(* CODESYS project TrabalhoFMSLadder.project

Project tree, tasks and I/O mapping:
  Device : CODESYS Control Win V3, 3S - Smart Software Solutions GmbH, order no. 305021, version 3.5.11.30
    application Application
      libraries: Standard, * (System); EA_XiocEvents, 3.5.2.0 (Eaton Automation); Standard64, * (System); Util, * (System)
      task MainTask (cyclic, interval t#20ms, priority 1) calls LinhaFabricacao, LinhaEntradaTampa, RobosDaora, LinhaSaidaUsinagem, EstacaoTampa, Armazenamento, SaidaPecas, EstacaoPallet
      Symbols
      program LinhaFabricacao [LD]
      program LinhaEntradaTampa [LD]
      program RobosDaora [LD]
      program LinhaSaidaUsinagem [LD]
      program EstacaoTampa [LD]
      program Armazenamento [LD]
      program SaidaPecas [LD]
      program EstacaoPallet [LD]
      program Teste [LD]
  program PLC_PRG_1 [LD]
  program PLC_PRG [LD]
  program PLC_PRG_2 [LD]
*)

// Device/Application/LinhaFabricacao
PROGRAM LinhaFabricacao
VAR
		//ENTRADAS
	SensorDifuso1CLP:BOOL;
	SensorDifuso2CLP:BOOL;
	VisionSensor1CLP:BOOL;
	VisionSensor2CLP:BOOL;
	ConveyorGate1OpenCLP:BOOL;
	
	//Saidas
	StopBlade1CLP:BOOL;
	StopBlade2CLP:BOOL;
	Pusher1CLP:BOOL;
	Pusher2CLP:BOOL;
	ConveyorGate1CLP:BOOL;
	Conveyor6m1CLP:BOOL;
	Conveyor6m2CLP:BOOL;
	
	
	//Memórias
	Conv6m1Vazio:BOOL;
	Conv6m2Vazio:BOOL;
	TravaVerde:BOOL;
	TravaAzul:BOOL;
	LerVerde: BOOL;
	LerAzul: BOOL;
	RejeitadoVerde:BOOL;
	RejeitadoAzul:BOOL;
	
	//vars timers
	ElapsedTime: TIME;
	ElapsedTime2: TIME;
	TimerVerde: TON;
	TimerAzul: TON;
	TimerPusher1: TON;
	TimerPusher2: TON;
END_VAR
VAR // added by the converter: edge detectors and wires of the graphical bodies
    _w1, _w2 : BOOL;
END_VAR

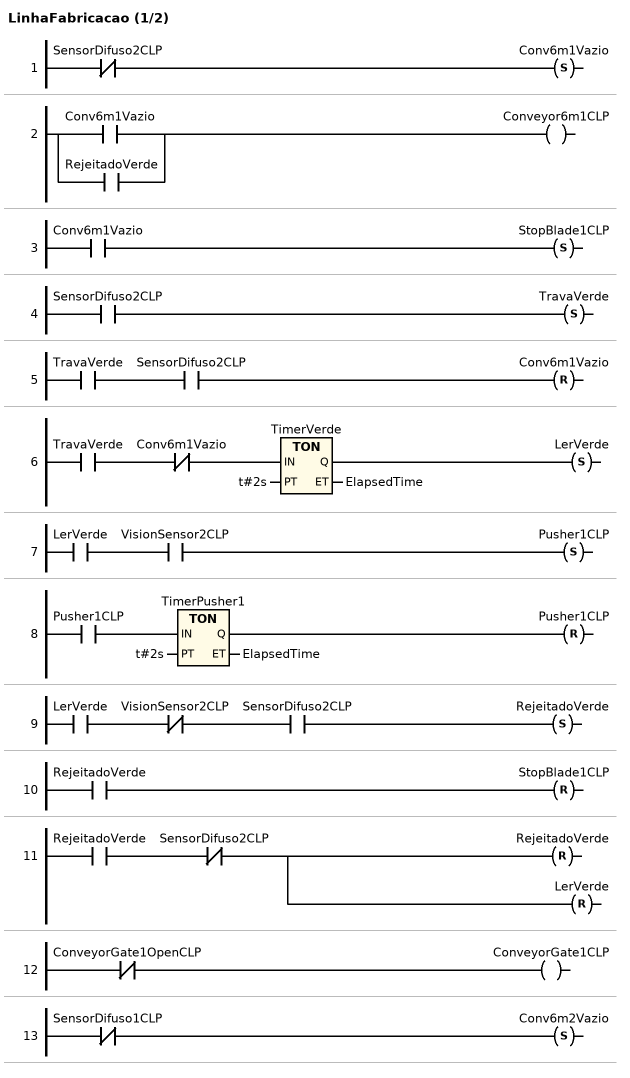
// NETWORK 1
Conv6m1Vazio S= NOT SensorDifuso2CLP;

// NETWORK 2
Conveyor6m1CLP := Conv6m1Vazio OR RejeitadoVerde;

// NETWORK 3
StopBlade1CLP S= Conv6m1Vazio;

// NETWORK 4
TravaVerde S= SensorDifuso2CLP;

// NETWORK 5
Conv6m1Vazio R= TravaVerde AND SensorDifuso2CLP;

// NETWORK 6
TimerVerde(IN := TravaVerde AND NOT Conv6m1Vazio, PT := t#2s, ET => ElapsedTime); // TON
LerVerde S= TimerVerde.Q;

// NETWORK 7
Pusher1CLP S= LerVerde AND VisionSensor2CLP;

// NETWORK 8
TimerPusher1(IN := Pusher1CLP, PT := t#2s, ET => ElapsedTime); // TON
Pusher1CLP R= TimerPusher1.Q;

// NETWORK 9
RejeitadoVerde S= LerVerde AND NOT VisionSensor2CLP AND SensorDifuso2CLP;

// NETWORK 10
StopBlade1CLP R= RejeitadoVerde;

// NETWORK 11
_w1 := RejeitadoVerde AND NOT SensorDifuso2CLP;
RejeitadoVerde R= _w1;
LerVerde R= _w1;

// NETWORK 12
ConveyorGate1CLP := NOT ConveyorGate1OpenCLP;

// NETWORK 13
Conv6m2Vazio S= NOT SensorDifuso1CLP;

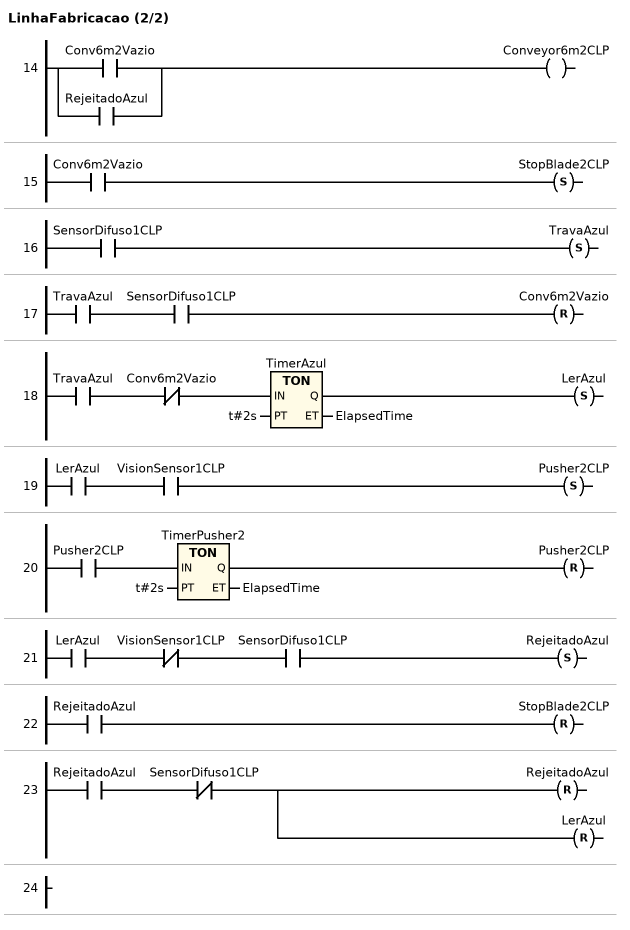
// NETWORK 14
Conveyor6m2CLP := Conv6m2Vazio OR RejeitadoAzul;

// NETWORK 15
StopBlade2CLP S= Conv6m2Vazio;

// NETWORK 16
TravaAzul S= SensorDifuso1CLP;

// NETWORK 17
Conv6m2Vazio R= TravaAzul AND SensorDifuso1CLP;

// NETWORK 18
TimerAzul(IN := TravaAzul AND NOT Conv6m2Vazio, PT := t#2s, ET => ElapsedTime); // TON
LerAzul S= TimerAzul.Q;

// NETWORK 19
Pusher2CLP S= LerAzul AND VisionSensor1CLP;

// NETWORK 20
TimerPusher2(IN := Pusher2CLP, PT := t#2s, ET => ElapsedTime); // TON
Pusher2CLP R= TimerPusher2.Q;

// NETWORK 21
RejeitadoAzul S= LerAzul AND NOT VisionSensor1CLP AND SensorDifuso1CLP;

// NETWORK 22
StopBlade2CLP R= RejeitadoAzul;

// NETWORK 23
_w2 := RejeitadoAzul AND NOT SensorDifuso1CLP;
RejeitadoAzul R= _w2;
LerAzul R= _w2;

// NETWORK 24

END_PROGRAM

// Device/Application/LinhaEntradaTampa
PROGRAM LinhaEntradaTampa
VAR
	//entradas
	VisionSensor3CLP:BOOL;
	SensorDifuso6CLP:BOOL;
	SensorDifuso7CLP:BOOL;
	
	//saidas
	Conveyor6m3CLP:BOOL;
	Conveyor4m1CLP:BOOL;
	ArmSorterCLP:BOOL;
	ArmBeltCLP:BOOL;
	Emmiter3CLP:BOOL;
	
	//memorias
	DivAzul:BOOL;
	TimerDiv: TON;
	Tempodiv: TIME;
	TimerDivR: TON;

	TesteCLP: BOOL;
	Nada: BOOL;
	StopBlade5CLP: BOOL;
	StopBlade6CLP: BOOL;
END_VAR

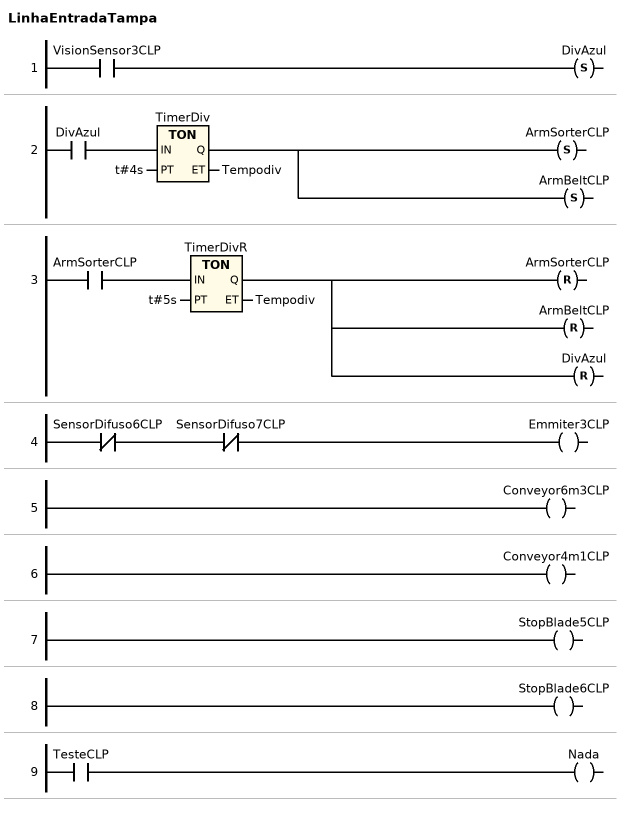
// NETWORK 1
DivAzul S= VisionSensor3CLP;

// NETWORK 2
TimerDiv(IN := DivAzul, PT := t#4s, ET => Tempodiv); // TON
ArmSorterCLP S= TimerDiv.Q;
ArmBeltCLP S= TimerDiv.Q;

// NETWORK 3
TimerDivR(IN := ArmSorterCLP, PT := t#5s, ET => Tempodiv); // TON
ArmSorterCLP R= TimerDivR.Q;
ArmBeltCLP R= TimerDivR.Q;
DivAzul R= TimerDivR.Q;

// NETWORK 4
Emmiter3CLP := NOT SensorDifuso6CLP AND NOT SensorDifuso7CLP;

// NETWORK 5
Conveyor6m3CLP := TRUE;

// NETWORK 6
Conveyor4m1CLP := TRUE;

// NETWORK 7
StopBlade5CLP := TRUE;

// NETWORK 8
StopBlade6CLP := TRUE;

// NETWORK 9
Nada := TesteCLP;

END_PROGRAM

// Device/Application/RobosDaora
PROGRAM RobosDaora
VAR
	//saidas
	MachinigCenter1StartCLP:BOOL;
	MachinigCenter2StartCLP:BOOL;
	MachinigCenter1StopCLP:BOOL;
	MachinigCenter2StopCLP:BOOL;
	MachinigCenter1ResetCLP:BOOL;
	MachinigCenter2ResetCLP:BOOL;

	//memorias
	InitialStart: TP;
	timepulse: TIME;
	BotaoSupLiga1:BOOL;
	BotaoSupLiga2:BOOL;
	BotaoSupPara1:BOOL;
	BotaoSupPara2:BOOL;
	BotaoSupReset1:BOOL;
	BotaoSupReset2:BOOL;
	
	//fb
	Progress1CLP: INT;
	Nada: BOOL;
	FDS1: INT;
	Progress2CLP: INT;
	FDS2: INT;
	Start1CLP: BOOL;
	Start2CLP: BOOL;
	Stop1CLP: BOOL;
	Stop2CLP: BOOL;
	Open1CLP: BOOL;
	Open2CLP: BOOL;
END_VAR

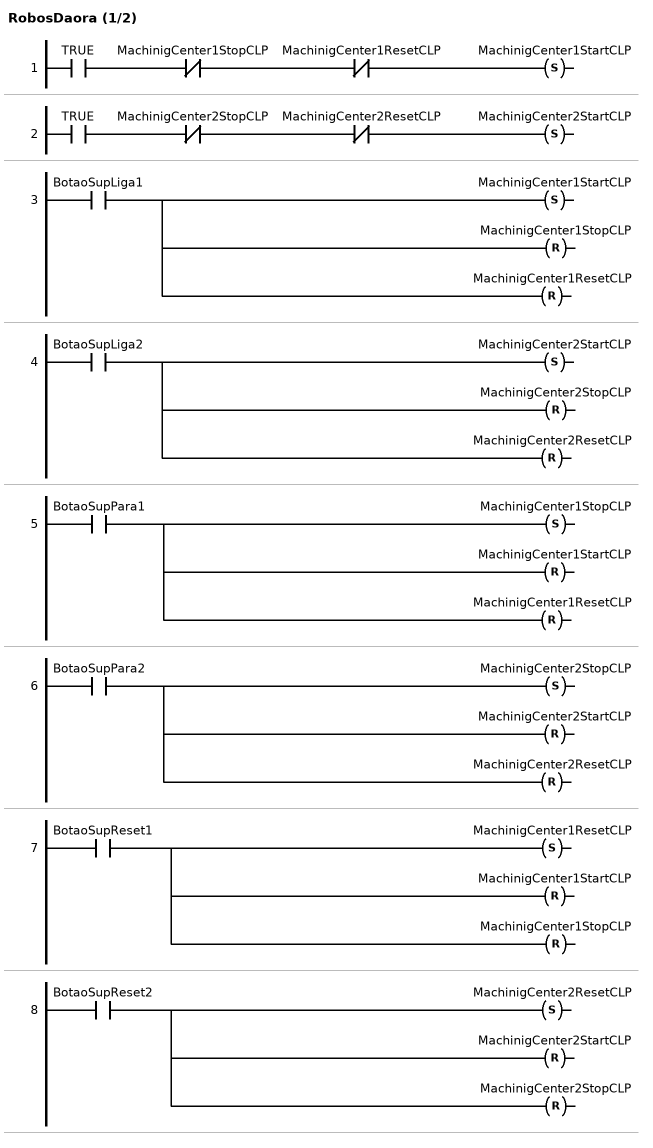
// NETWORK 1
MachinigCenter1StartCLP S= TRUE AND NOT MachinigCenter1StopCLP AND NOT MachinigCenter1ResetCLP;

// NETWORK 2
MachinigCenter2StartCLP S= TRUE AND NOT MachinigCenter2StopCLP AND NOT MachinigCenter2ResetCLP;

// NETWORK 3
MachinigCenter1StartCLP S= BotaoSupLiga1;
MachinigCenter1StopCLP R= BotaoSupLiga1;
MachinigCenter1ResetCLP R= BotaoSupLiga1;

// NETWORK 4
MachinigCenter2StartCLP S= BotaoSupLiga2;
MachinigCenter2StopCLP R= BotaoSupLiga2;
MachinigCenter2ResetCLP R= BotaoSupLiga2;

// NETWORK 5
MachinigCenter1StopCLP S= BotaoSupPara1;
MachinigCenter1StartCLP R= BotaoSupPara1;
MachinigCenter1ResetCLP R= BotaoSupPara1;

// NETWORK 6
MachinigCenter2StopCLP S= BotaoSupPara2;
MachinigCenter2StartCLP R= BotaoSupPara2;
MachinigCenter2ResetCLP R= BotaoSupPara2;

// NETWORK 7
MachinigCenter1ResetCLP S= BotaoSupReset1;
MachinigCenter1StartCLP R= BotaoSupReset1;
MachinigCenter1StopCLP R= BotaoSupReset1;

// NETWORK 8
MachinigCenter2ResetCLP S= BotaoSupReset2;
MachinigCenter2StartCLP R= BotaoSupReset2;
MachinigCenter2StopCLP R= BotaoSupReset2;

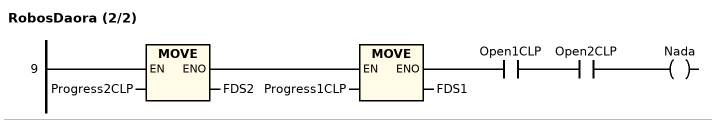
// NETWORK 9
FDS2 := Progress2CLP;
FDS1 := Progress1CLP;
Nada := Open1CLP AND Open2CLP;

END_PROGRAM

// Device/Application/LinhaSaidaUsinagem
PROGRAM LinhaSaidaUsinagem
VAR
	//SAIDAS
	EsteiraUsinada1CLP:BOOL;
	EsteiraPortaoUsinadaCLP:BOOL;
	Conveyor4m2CLP:BOOL;
	Conveyor2m1CLP:BOOL;
	StopBlade7CLP:BOOL;
	
	//ENTRADAS
	SensorDifuso5CLP:BOOL;
	PortaoUsinadaOpenCLP:BOOL;
	
	//Memórias
	EsteirasON:BOOL;
	PecaDentro:BOOL;
	PecaNoSensor:BOOL;
END_VAR
VAR // added by the converter: edge detectors and wires of the graphical bodies
    _w1, _w2 : BOOL;
END_VAR

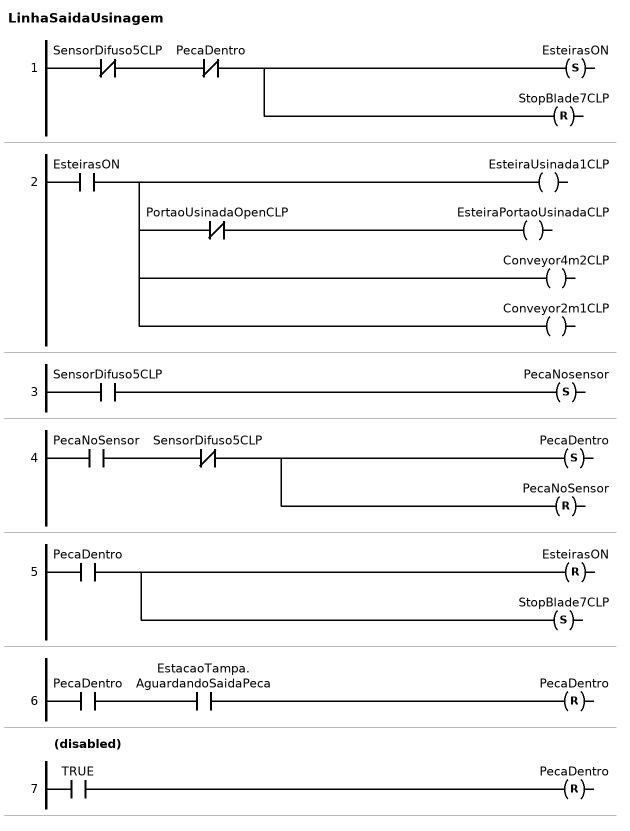
// NETWORK 1
_w1 := NOT SensorDifuso5CLP AND NOT PecaDentro;
EsteirasON S= _w1;
StopBlade7CLP R= _w1;

// NETWORK 2
EsteiraUsinada1CLP := EsteirasON;
EsteiraPortaoUsinadaCLP := EsteirasON AND NOT PortaoUsinadaOpenCLP;
Conveyor4m2CLP := EsteirasON;
Conveyor2m1CLP := EsteirasON;

// NETWORK 3
PecaNosensor S= SensorDifuso5CLP;

// NETWORK 4
_w2 := PecaNoSensor AND NOT SensorDifuso5CLP;
PecaDentro S= _w2;
PecaNoSensor R= _w2;

// NETWORK 5
EsteirasON R= PecaDentro;
StopBlade7CLP S= PecaDentro;

// NETWORK 6
PecaDentro R= PecaDentro AND EstacaoTampa.AguardandoSaidaPeca;

// NETWORK 7 (disabled)
// PecaDentro R= TRUE;

END_PROGRAM

// Device/Application/EstacaoTampa
PROGRAM EstacaoTampa
VAR
	//SAIDAS
	Conveyor2m3CLP:BOOL;
	StopBlade4CLP:BOOL;
	Pick1XSetPointCLP:LREAL;
	Pick1YSetPointCLP:LREAL;
	Pick1ZSetPointCLP:LREAL;
	Pick1GrabCLP:BOOL;
	//ENTRADAS
	PickSensorCLP:BOOL;
	VisionSensor4_0CLP:BOOL;
	VisionSensor4_1CLP:BOOL;
	VisionSensor4_2CLP:BOOL;
	
	//MEMORIAS
	EsteiraON:BOOL;
	VerCor:BOOL;
	PegaAzul:BOOL;
	PegaVerde:BOOL;
	AvancaTampa:BOOL;
	PegaTampa:BOOL;
	RecuaGraber:BOOL;
	GraberRecuado:BOOL;
	TampaPegada:BOOL;
	ColetaTampa:BOOL;
	ColocarTampa:BOOL;
	TampaPosicionada:BOOL;
	SoltaTampa:BOOL;
	PosicaoDescanso:BOOL;
	RetornoPosInicial:BOOL;
	LiberarPeca:BOOL;
	AguardandoSaidaPeca:BOOL;
	EstacaoOcupada:BOOL;
	
	TimerMove1: TON;
	ElapsedTime1: TIME;
	TimerPegar: TON;
	ElapsedTime2: TIME;
	TimerRecuo: TON;
	TimerMove2: TON;
	TimerWait: TON;
	ElapsedTime3: TIME;
	ElapsedTime4: TIME;
	ElapsedTime5: TIME;
	ElapsedTime6: TIME;
	ElapsedTIme7: TIME;
	TimerRecuo2: TON;
	TimerMove3: TON;
	TimerSoltar: TON;
	ElapsedTime8: TIME;
	TimerSaida: TON;
	ElapsedTime9: TIME;
	TimerWait2: TON;
	ElapsedTIme10: TIME;
	TimerWait3: TON;
	ElapsedTime11: TIME;
END_VAR
VAR // added by the converter: edge detectors and wires of the graphical bodies
    _w1, _w2, _w3, _w4, _w5, _w6, _w7, _w8, _w9, _w10, _w11, _w12 : BOOL;
END_VAR

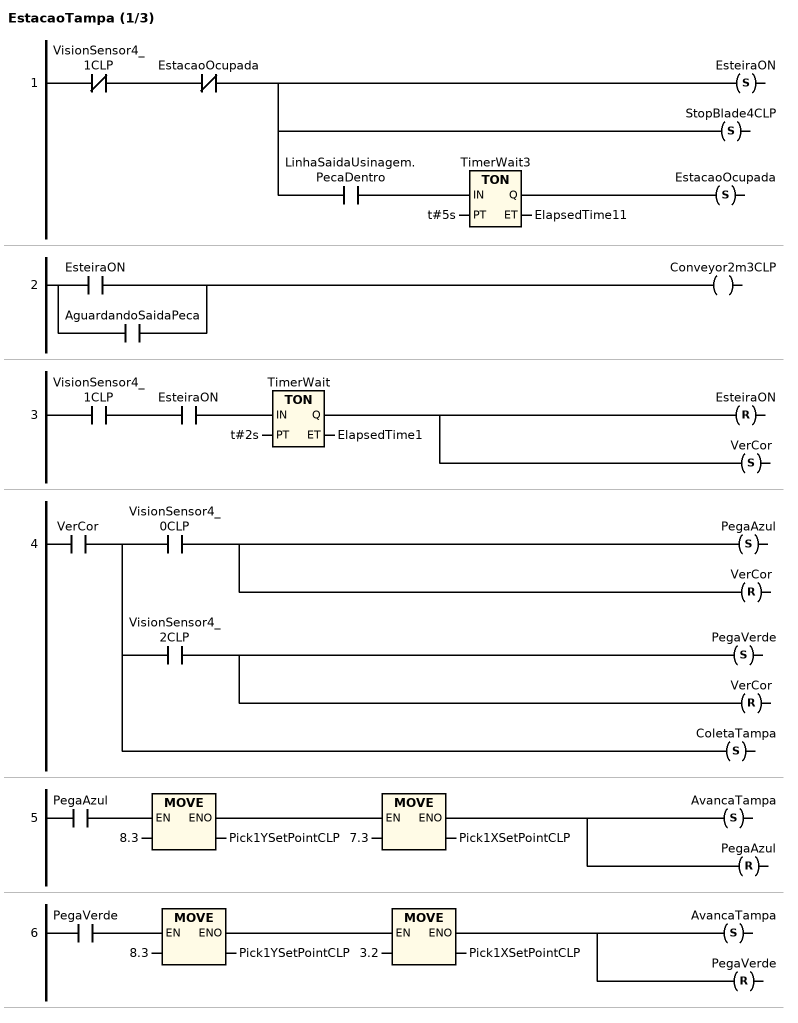
// NETWORK 1
_w1 := NOT VisionSensor4_1CLP AND NOT EstacaoOcupada;
EsteiraON S= _w1;
StopBlade4CLP S= _w1;
TimerWait3(IN := _w1 AND LinhaSaidaUsinagem.PecaDentro, PT := t#5s, ET => ElapsedTime11); // TON
EstacaoOcupada S= TimerWait3.Q;

// NETWORK 2
Conveyor2m3CLP := EsteiraON OR AguardandoSaidaPeca;

// NETWORK 3
TimerWait(IN := VisionSensor4_1CLP AND EsteiraON, PT := t#2s, ET => ElapsedTime1); // TON
EsteiraON R= TimerWait.Q;
VerCor S= TimerWait.Q;

// NETWORK 4
_w2 := VerCor;
_w3 := _w2 AND VisionSensor4_0CLP;
PegaAzul S= _w3;
VerCor R= _w3;
_w4 := _w2 AND VisionSensor4_2CLP;
PegaVerde S= _w4;
VerCor R= _w4;
ColetaTampa S= _w2;

// NETWORK 5
_w5 := PegaAzul;
IF _w5 THEN Pick1YSetPointCLP := 8.3; END_IF
IF _w5 THEN Pick1XSetPointCLP := 7.3; END_IF
AvancaTampa S= _w5;
PegaAzul R= _w5;

// NETWORK 6
_w6 := PegaVerde;
IF _w6 THEN Pick1YSetPointCLP := 8.3; END_IF
IF _w6 THEN Pick1XSetPointCLP := 3.2; END_IF
AvancaTampa S= _w6;
PegaVerde R= _w6;

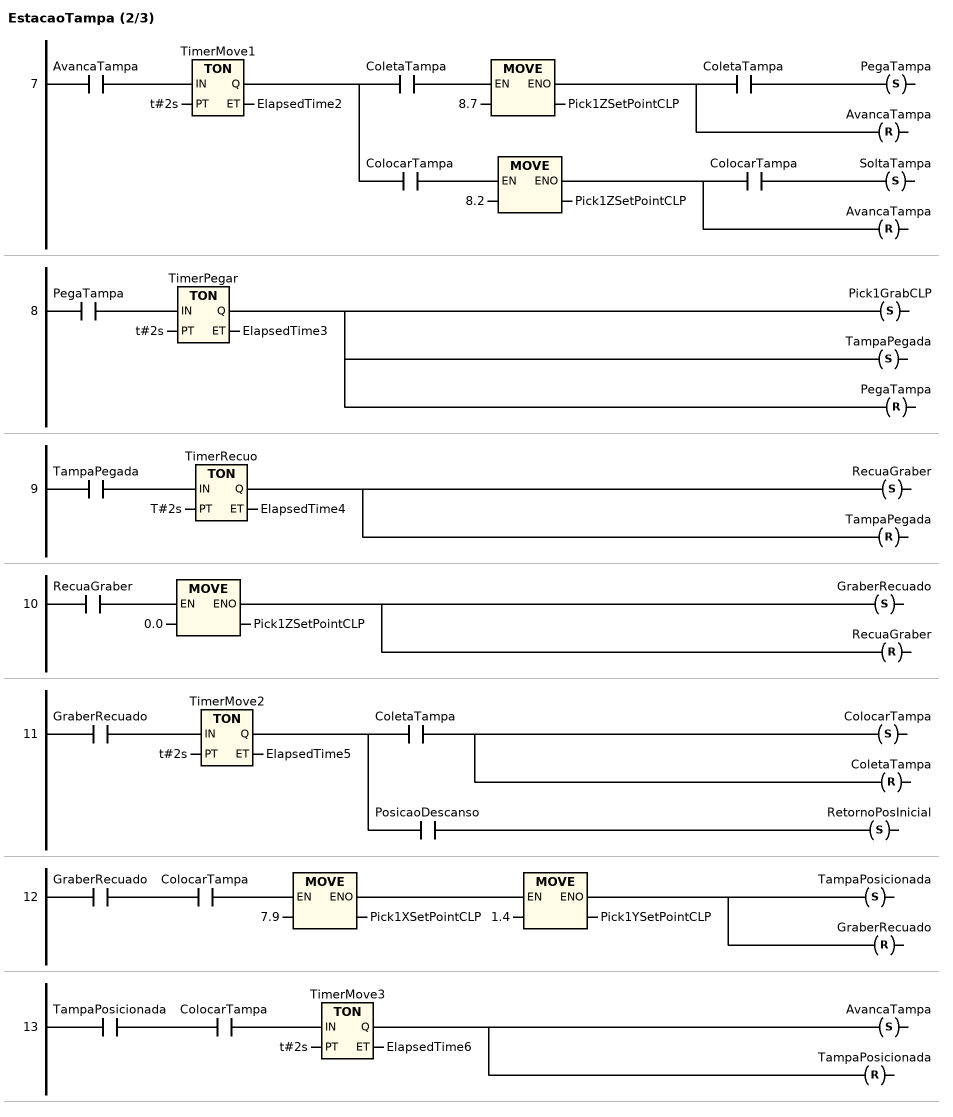
// NETWORK 7
TimerMove1(IN := AvancaTampa, PT := t#2s, ET => ElapsedTime2); // TON
_w7 := TimerMove1.Q AND ColetaTampa;
IF _w7 THEN Pick1ZSetPointCLP := 8.7; END_IF
PegaTampa S= _w7 AND ColetaTampa;
AvancaTampa R= _w7;
_w8 := TimerMove1.Q AND ColocarTampa;
IF _w8 THEN Pick1ZSetPointCLP := 8.2; END_IF
SoltaTampa S= _w8 AND ColocarTampa;
AvancaTampa R= _w8;

// NETWORK 8
TimerPegar(IN := PegaTampa, PT := t#2s, ET => ElapsedTime3); // TON
Pick1GrabCLP S= TimerPegar.Q;
TampaPegada S= TimerPegar.Q;
PegaTampa R= TimerPegar.Q;

// NETWORK 9
TimerRecuo(IN := TampaPegada, PT := T#2s, ET => ElapsedTime4); // TON
RecuaGraber S= TimerRecuo.Q;
TampaPegada R= TimerRecuo.Q;

// NETWORK 10
_w9 := RecuaGraber;
IF _w9 THEN Pick1ZSetPointCLP := 0.0; END_IF
GraberRecuado S= _w9;
RecuaGraber R= _w9;

// NETWORK 11
TimerMove2(IN := GraberRecuado, PT := t#2s, ET => ElapsedTime5); // TON
_w10 := TimerMove2.Q AND ColetaTampa;
ColocarTampa S= _w10;
ColetaTampa R= _w10;
RetornoPosInicial S= TimerMove2.Q AND PosicaoDescanso;

// NETWORK 12
_w11 := GraberRecuado AND ColocarTampa;
IF _w11 THEN Pick1XSetPointCLP := 7.9; END_IF
IF _w11 THEN Pick1YSetPointCLP := 1.4; END_IF
TampaPosicionada S= _w11;
GraberRecuado R= _w11;

// NETWORK 13
TimerMove3(IN := TampaPosicionada AND ColocarTampa, PT := t#2s, ET => ElapsedTime6); // TON
AvancaTampa S= TimerMove3.Q;
TampaPosicionada R= TimerMove3.Q;

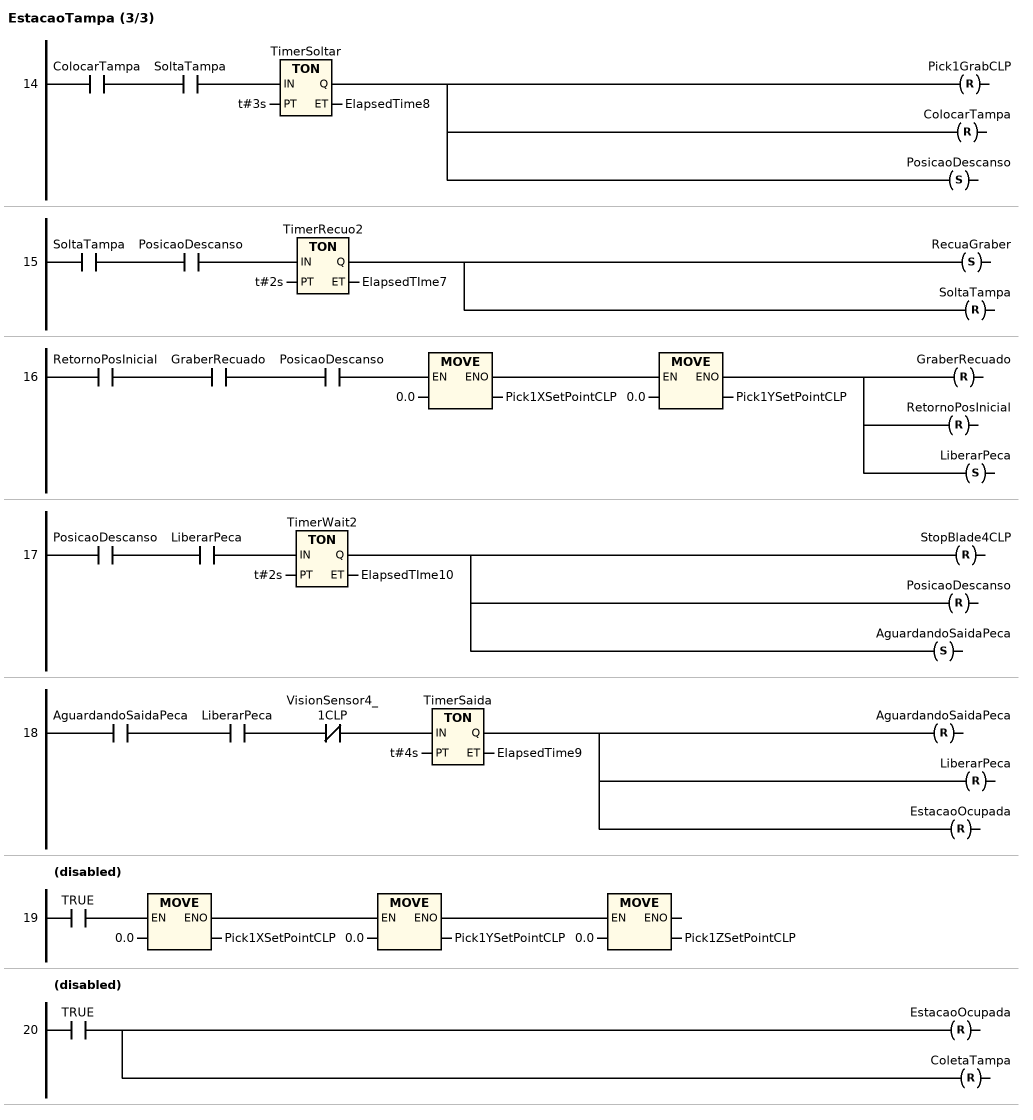
// NETWORK 14
TimerSoltar(IN := ColocarTampa AND SoltaTampa, PT := t#3s, ET => ElapsedTime8); // TON
Pick1GrabCLP R= TimerSoltar.Q;
ColocarTampa R= TimerSoltar.Q;
PosicaoDescanso S= TimerSoltar.Q;

// NETWORK 15
TimerRecuo2(IN := SoltaTampa AND PosicaoDescanso, PT := t#2s, ET => ElapsedTIme7); // TON
RecuaGraber S= TimerRecuo2.Q;
SoltaTampa R= TimerRecuo2.Q;

// NETWORK 16
_w12 := RetornoPosInicial AND GraberRecuado AND PosicaoDescanso;
IF _w12 THEN Pick1XSetPointCLP := 0.0; END_IF
IF _w12 THEN Pick1YSetPointCLP := 0.0; END_IF
GraberRecuado R= _w12;
RetornoPosInicial R= _w12;
LiberarPeca S= _w12;

// NETWORK 17
TimerWait2(IN := PosicaoDescanso AND LiberarPeca, PT := t#2s, ET => ElapsedTIme10); // TON
StopBlade4CLP R= TimerWait2.Q;
PosicaoDescanso R= TimerWait2.Q;
AguardandoSaidaPeca S= TimerWait2.Q;

// NETWORK 18
TimerSaida(
    IN := AguardandoSaidaPeca AND LiberarPeca AND NOT VisionSensor4_1CLP,
    PT := t#4s,
    ET => ElapsedTime9); // TON
AguardandoSaidaPeca R= TimerSaida.Q;
LiberarPeca R= TimerSaida.Q;
EstacaoOcupada R= TimerSaida.Q;

// NETWORK 19 (disabled)
// Pick1XSetPointCLP := 0.0;
// Pick1YSetPointCLP := 0.0;
// Pick1ZSetPointCLP := 0.0;

// NETWORK 20 (disabled)
// EstacaoOcupada R= TRUE;
// ColetaTampa R= TRUE;

END_PROGRAM

// Device/Application/Armazenamento
PROGRAM Armazenamento
VAR
	//SAIDAS
	EntryConveyorCLP:BOOL;
	LoadCOnveyorCLP:BOOL;
	ForksRightCLP:BOOL;
	ForksLeftCLP:BOOL;
	ForkLiftCLP:BOOL;
	TargetPositionCLP:INT;
	UnloadConveyorCLP:BOOL;
	//Entradas
	AtEntrySensorCLP:BOOL;
	AtLoadSensorCLP:BOOL;
	AtMiddleSensorCLP:BOOL;
	AtUnloadSensorCLP:BOOL;
	MovingXCLP:BOOL;
	
	//Memorias
	EntryConveyorOcupado:BOOL;
	PalletSensorEntrada: BOOL;
	LoadConveyorOcupado: BOOL;
	InicioCarregamento: BOOL;
	GarfoLoad: BOOL;
	GarfoLiftLoad: BOOL;
	FaseCarregamento: BOOL;
	PalletCarregado: BOOL;
	PalletsDentro: WORD;
	IndoDestinoCarga: BOOL;
	LocalDestinoCarga: BOOL;
	GarfoPalletArmazem: BOOL;
	RetornarPosiDescanso: BOOL;
	PalletColocado: BOOL;
	RetronandoPosDescanso: BOOL;
	DescargaHabilitado: BOOL;
	InicioDescarga: BOOL;
	FaseDescarga: BOOL;
	IndoPosDescarga: BOOL;
	PosDescarga: BOOL;
	GarfoDesArmazem: BOOL;
	GarfoDesErguido: BOOL;
	PalletRetirado: BOOL;
	RetornarPosDescarga: BOOL;
	RetornandoPosDescarga: BOOL;
	PosSaida: BOOL;
	PalletAcimaSaida: BOOL;
	PalletNaSaida: BOOL;
	DescargaFeita: BOOL;
	
	Timer1: TON;
	ElapsedTime1: TIME;
	TimerCount: TP;
	ElapsedTime2: TIME;
	AUmentaPallet: CTU;
	TimerWait2: TON;
	TimerWait3: TON;
	ElapsedTime3: TIME;
	TimerWait4: TON;
	ElapsedTime4: TIME;
	TimerWait5: TON;
	ElapsedTime5: TIME;
	TimerWait6: TON;
	ElapsedTime6: TIME;
	TimerWait7: TON;
	ElapsedTime7: TIME;
	TimerWait8: TON;
	ElapsedTime8: TIME;
	TimerWait9: TON;
	ElapsedTime9: TIME;	
	TimerWait10: TON;
	ElapsedTime10: TIME;
	TimerWait11: TON;
	ElapsedTime11: TIME;	
	TimerWait12: TON;
	ElapsedTime12: TIME;
	TimerCount2: TP;
	ElapsedCount2: TIME;
	DiminuiPallet: CTD;
	TimerWait13: TON;
	ElapsedTime13: TIME;
	TimerWait14: TON;
	ElapsedTime14: TIME;
	TimerWait15: TON;
	ElapsedTime15: TIME;
	QntidadePallets: WORD;
END_VAR
VAR // added by the converter: edge detectors and wires of the graphical bodies
    _w1, _w2, _w3, _w4, _w5, _w6, _w7, _w8, _w9, _w10, _w11, _w12 : BOOL;
END_VAR

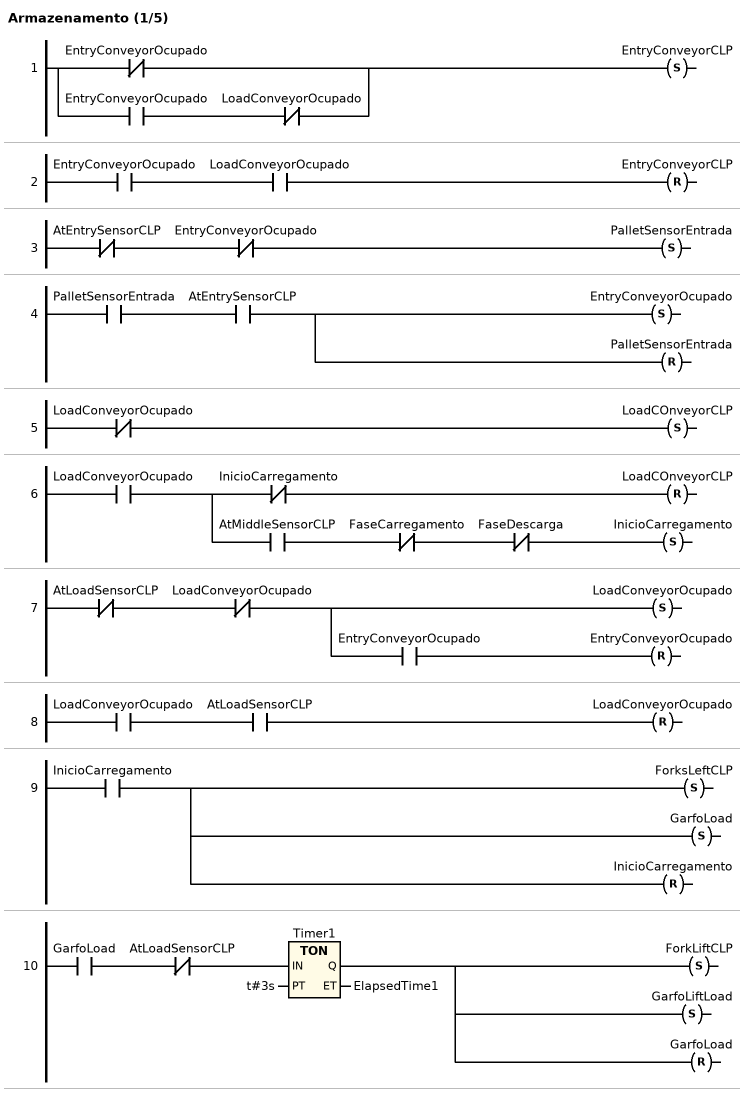
// NETWORK 1
EntryConveyorCLP S= NOT EntryConveyorOcupado OR EntryConveyorOcupado AND NOT LoadConveyorOcupado;

// NETWORK 2
EntryConveyorCLP R= EntryConveyorOcupado AND LoadConveyorOcupado;

// NETWORK 3
PalletSensorEntrada S= NOT AtEntrySensorCLP AND NOT EntryConveyorOcupado;

// NETWORK 4
_w1 := PalletSensorEntrada AND AtEntrySensorCLP;
EntryConveyorOcupado S= _w1;
PalletSensorEntrada R= _w1;

// NETWORK 5
LoadCOnveyorCLP S= NOT LoadConveyorOcupado;

// NETWORK 6
LoadCOnveyorCLP R= LoadConveyorOcupado AND NOT InicioCarregamento;
InicioCarregamento S= LoadConveyorOcupado AND AtMiddleSensorCLP AND NOT FaseCarregamento AND NOT FaseDescarga;

// NETWORK 7
_w2 := NOT AtLoadSensorCLP AND NOT LoadConveyorOcupado;
LoadConveyorOcupado S= _w2;
EntryConveyorOcupado R= _w2 AND EntryConveyorOcupado;

// NETWORK 8
LoadConveyorOcupado R= LoadConveyorOcupado AND AtLoadSensorCLP;

// NETWORK 9
_w3 := InicioCarregamento;
ForksLeftCLP S= _w3;
GarfoLoad S= _w3;
InicioCarregamento R= _w3;

// NETWORK 10
Timer1(IN := GarfoLoad AND NOT AtLoadSensorCLP, PT := t#3s, ET => ElapsedTime1); // TON
ForkLiftCLP S= Timer1.Q;
GarfoLiftLoad S= Timer1.Q;
GarfoLoad R= Timer1.Q;

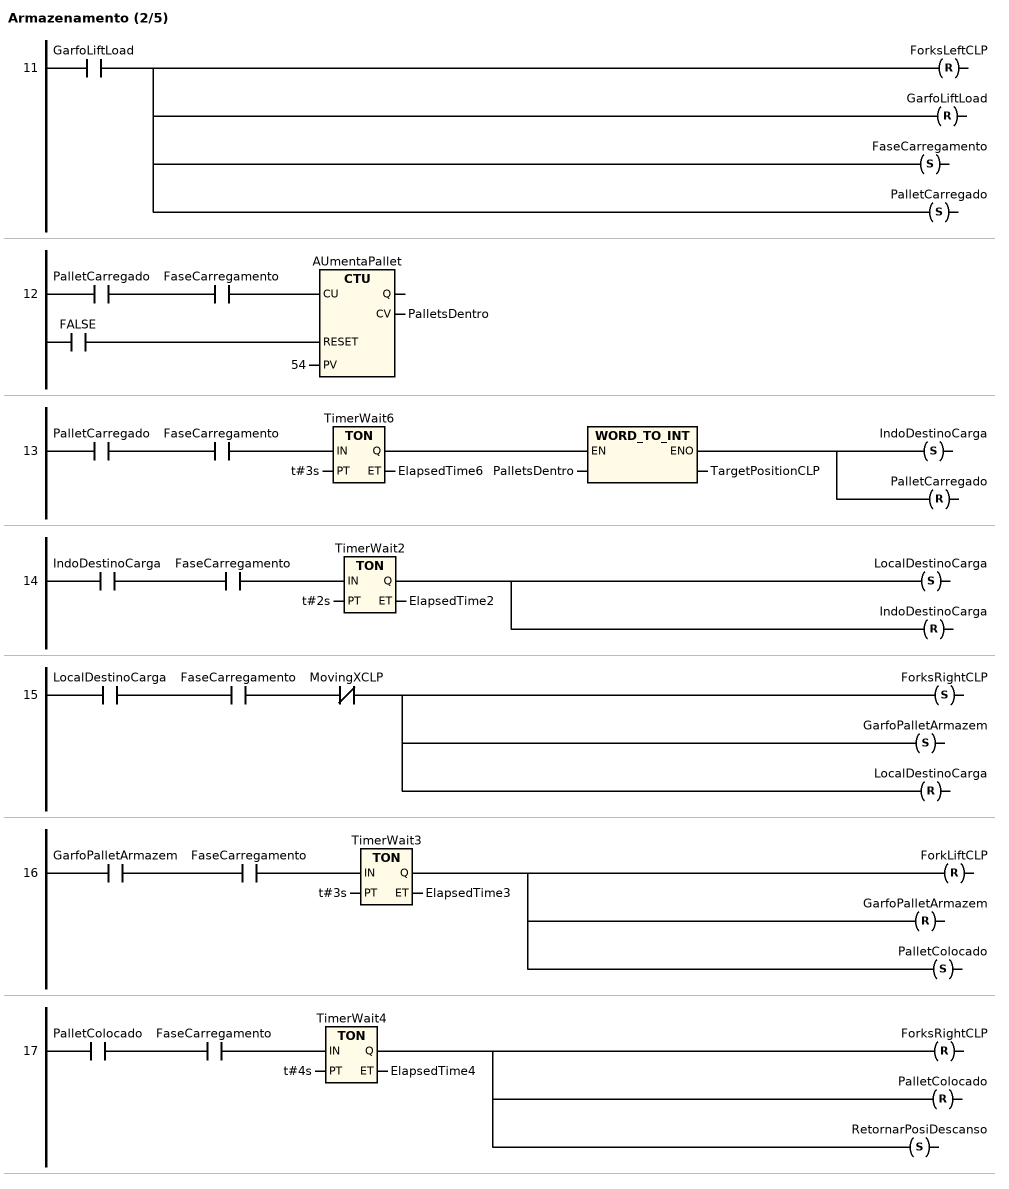
// NETWORK 11
_w4 := GarfoLiftLoad;
ForksLeftCLP R= _w4;
GarfoLiftLoad R= _w4;
FaseCarregamento S= _w4;
PalletCarregado S= _w4;

// NETWORK 12
AUmentaPallet(CU := PalletCarregado AND FaseCarregamento, RESET := FALSE, PV := 54, CV => PalletsDentro); // CTU

// NETWORK 13
TimerWait6(IN := PalletCarregado AND FaseCarregamento, PT := t#3s, ET => ElapsedTime6); // TON
_w5 := TimerWait6.Q;
IF _w5 THEN TargetPositionCLP := WORD_TO_INT(PalletsDentro); END_IF
IndoDestinoCarga S= _w5;
PalletCarregado R= _w5;

// NETWORK 14
TimerWait2(IN := IndoDestinoCarga AND FaseCarregamento, PT := t#2s, ET => ElapsedTime2); // TON
LocalDestinoCarga S= TimerWait2.Q;
IndoDestinoCarga R= TimerWait2.Q;

// NETWORK 15
_w6 := LocalDestinoCarga AND FaseCarregamento AND NOT MovingXCLP;
ForksRightCLP S= _w6;
GarfoPalletArmazem S= _w6;
LocalDestinoCarga R= _w6;

// NETWORK 16
TimerWait3(IN := GarfoPalletArmazem AND FaseCarregamento, PT := t#3s, ET => ElapsedTime3); // TON
ForkLiftCLP R= TimerWait3.Q;
GarfoPalletArmazem R= TimerWait3.Q;
PalletColocado S= TimerWait3.Q;

// NETWORK 17
TimerWait4(IN := PalletColocado AND FaseCarregamento, PT := t#4s, ET => ElapsedTime4); // TON
ForksRightCLP R= TimerWait4.Q;
PalletColocado R= TimerWait4.Q;
RetornarPosiDescanso S= TimerWait4.Q;

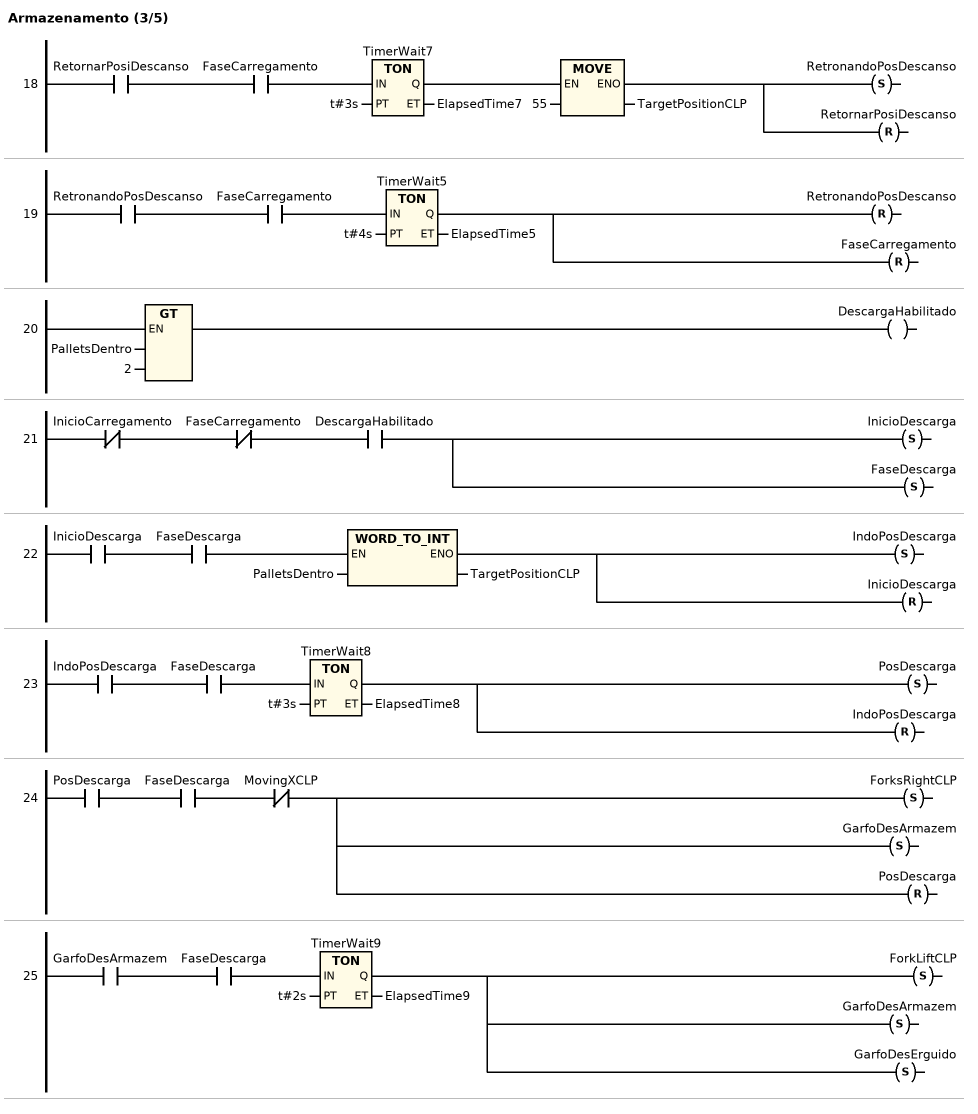
// NETWORK 18
TimerWait7(IN := RetornarPosiDescanso AND FaseCarregamento, PT := t#3s, ET => ElapsedTime7); // TON
_w7 := TimerWait7.Q;
IF _w7 THEN TargetPositionCLP := 55; END_IF
RetronandoPosDescanso S= _w7;
RetornarPosiDescanso R= _w7;

// NETWORK 19
TimerWait5(IN := RetronandoPosDescanso AND FaseCarregamento, PT := t#4s, ET => ElapsedTime5); // TON
RetronandoPosDescanso R= TimerWait5.Q;
FaseCarregamento R= TimerWait5.Q;

// NETWORK 20
DescargaHabilitado := PalletsDentro > 2;

// NETWORK 21
_w8 := NOT InicioCarregamento AND NOT FaseCarregamento AND DescargaHabilitado;
InicioDescarga S= _w8;
FaseDescarga S= _w8;

// NETWORK 22
_w9 := InicioDescarga AND FaseDescarga;
IF _w9 THEN TargetPositionCLP := WORD_TO_INT(PalletsDentro); END_IF
IndoPosDescarga S= _w9;
InicioDescarga R= _w9;

// NETWORK 23
TimerWait8(IN := IndoPosDescarga AND FaseDescarga, PT := t#3s, ET => ElapsedTime8); // TON
PosDescarga S= TimerWait8.Q;
IndoPosDescarga R= TimerWait8.Q;

// NETWORK 24
_w10 := PosDescarga AND FaseDescarga AND NOT MovingXCLP;
ForksRightCLP S= _w10;
GarfoDesArmazem S= _w10;
PosDescarga R= _w10;

// NETWORK 25
TimerWait9(IN := GarfoDesArmazem AND FaseDescarga, PT := t#2s, ET => ElapsedTime9); // TON
ForkLiftCLP S= TimerWait9.Q;
GarfoDesArmazem S= TimerWait9.Q;
GarfoDesErguido S= TimerWait9.Q;

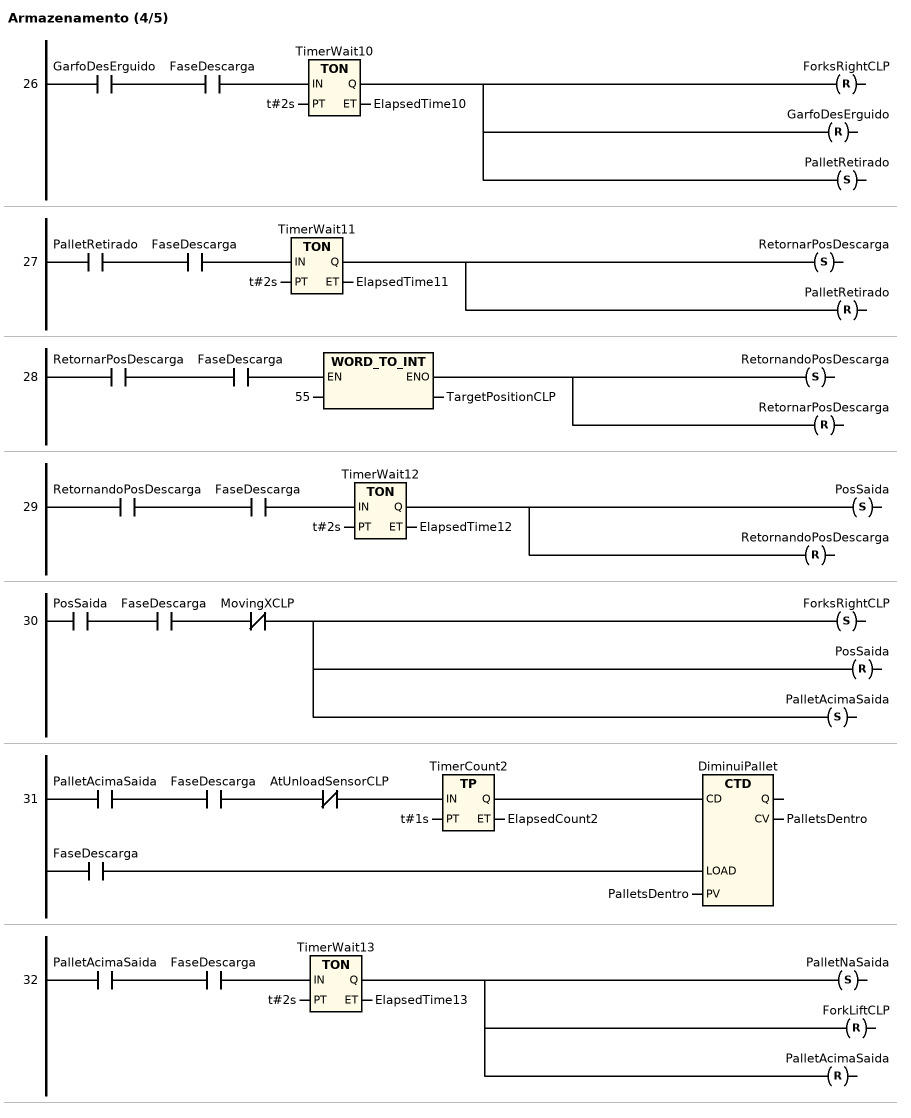
// NETWORK 26
TimerWait10(IN := GarfoDesErguido AND FaseDescarga, PT := t#2s, ET => ElapsedTime10); // TON
ForksRightCLP R= TimerWait10.Q;
GarfoDesErguido R= TimerWait10.Q;
PalletRetirado S= TimerWait10.Q;

// NETWORK 27
TimerWait11(IN := PalletRetirado AND FaseDescarga, PT := t#2s, ET => ElapsedTime11); // TON
RetornarPosDescarga S= TimerWait11.Q;
PalletRetirado R= TimerWait11.Q;

// NETWORK 28
_w11 := RetornarPosDescarga AND FaseDescarga;
IF _w11 THEN TargetPositionCLP := WORD_TO_INT(55); END_IF
RetornandoPosDescarga S= _w11;
RetornarPosDescarga R= _w11;

// NETWORK 29
TimerWait12(IN := RetornandoPosDescarga AND FaseDescarga, PT := t#2s, ET => ElapsedTime12); // TON
PosSaida S= TimerWait12.Q;
RetornandoPosDescarga R= TimerWait12.Q;

// NETWORK 30
_w12 := PosSaida AND FaseDescarga AND NOT MovingXCLP;
ForksRightCLP S= _w12;
PosSaida R= _w12;
PalletAcimaSaida S= _w12;

// NETWORK 31
TimerCount2(
    IN := PalletAcimaSaida AND FaseDescarga AND NOT AtUnloadSensorCLP,
    PT := t#1s,
    ET => ElapsedCount2); // TP
DiminuiPallet(CD := TimerCount2.Q, LOAD := FaseDescarga, PV := PalletsDentro, CV => PalletsDentro); // CTD

// NETWORK 32
TimerWait13(IN := PalletAcimaSaida AND FaseDescarga, PT := t#2s, ET => ElapsedTime13); // TON
PalletNaSaida S= TimerWait13.Q;
ForkLiftCLP R= TimerWait13.Q;
PalletAcimaSaida R= TimerWait13.Q;

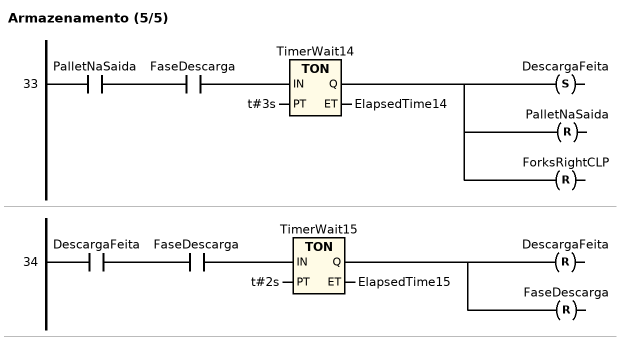
// NETWORK 33
TimerWait14(IN := PalletNaSaida AND FaseDescarga, PT := t#3s, ET => ElapsedTime14); // TON
DescargaFeita S= TimerWait14.Q;
PalletNaSaida R= TimerWait14.Q;
ForksRightCLP R= TimerWait14.Q;

// NETWORK 34
TimerWait15(IN := DescargaFeita AND FaseDescarga, PT := t#2s, ET => ElapsedTime15); // TON
DescargaFeita R= TimerWait15.Q;
FaseDescarga R= TimerWait15.Q;

END_PROGRAM

// Device/Application/SaidaPecas
PROGRAM SaidaPecas
VAR
	RollerConveyot2m2CLP: BOOL;
	VisionSensor5CLP: BOOL;
	azul: BOOL;
	TunableBackLimitCLP: BOOL;
	TunableRollmaisCLP: BOOL;
	TunableFrontLimitCLP: BOOL;
	TunableTurnCLP: BOOL;
	TON_0: TON;
	time_1: TIME;
	descarregar: BOOL;
	TON_1: TON;
	time_2: TIME;
END_VAR

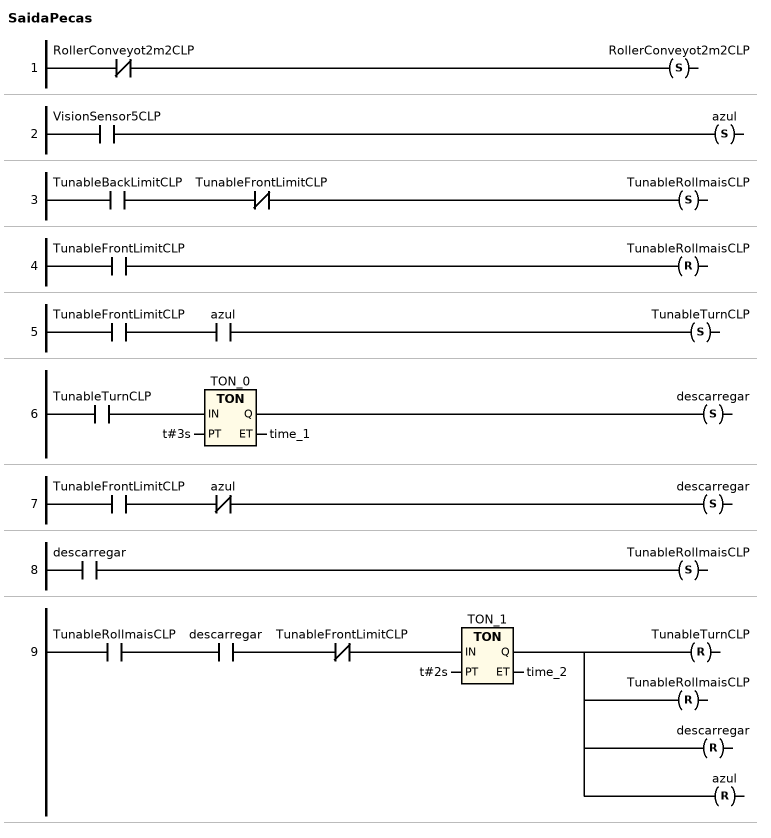
// NETWORK 1
RollerConveyot2m2CLP S= NOT RollerConveyot2m2CLP;

// NETWORK 2
azul S= VisionSensor5CLP;

// NETWORK 3
TunableRollmaisCLP S= TunableBackLimitCLP AND NOT TunableFrontLimitCLP;

// NETWORK 4
TunableRollmaisCLP R= TunableFrontLimitCLP;

// NETWORK 5
TunableTurnCLP S= TunableFrontLimitCLP AND azul;

// NETWORK 6
TON_0(IN := TunableTurnCLP, PT := t#3s, ET => time_1); // TON
descarregar S= TON_0.Q;

// NETWORK 7
descarregar S= TunableFrontLimitCLP AND NOT azul;

// NETWORK 8
TunableRollmaisCLP S= descarregar;

// NETWORK 9
TON_1(IN := TunableRollmaisCLP AND descarregar AND NOT TunableFrontLimitCLP, PT := t#2s, ET => time_2); // TON
TunableTurnCLP R= TON_1.Q;
TunableRollmaisCLP R= TON_1.Q;
descarregar R= TON_1.Q;
azul R= TON_1.Q;

END_PROGRAM

// Device/Application/EstacaoPallet
PROGRAM EstacaoPallet
VAR
	passando: BOOL;
	diffuse_sensor_3_clp: BOOL;
	passou: BOOL;
	two_axis_pick_z_clp: BOOL;
	two_axis_pick_x_clp: BOOL;
	TON_0: TON;
	time_1: TIME;
	two_axis_grab_clp: BOOL;
	TON_1: TON;
	time_2: TIME;
	carregado: BOOL;
	segunda_etapa: BOOL;
	TON_2: TON;
	time_3: TIME;
	TON_3: TON;
	time_4: TIME;
	TON_4: TON;
	time_5: TIME;
	voltar: BOOL;
	primeira_etapa: BOOL;
	TON_5: TON;
	time_6: TIME;
	pallet: BOOL;
	chain_tranfer_mais_1_clp: BOOL;
	diffuse_sensor_4_clp: BOOL;
	chain_transfer_left_clp: BOOL;
	TON_6: TON;
	time_7: TIME;
	rollet_conveyor_2m5CLP: BOOL;
	belt_conveyor_4m3_clp: BOOL;
END_VAR
VAR // added by the converter: edge detectors and wires of the graphical bodies
    _w1, _w2, _w3, _w4 : BOOL;
END_VAR

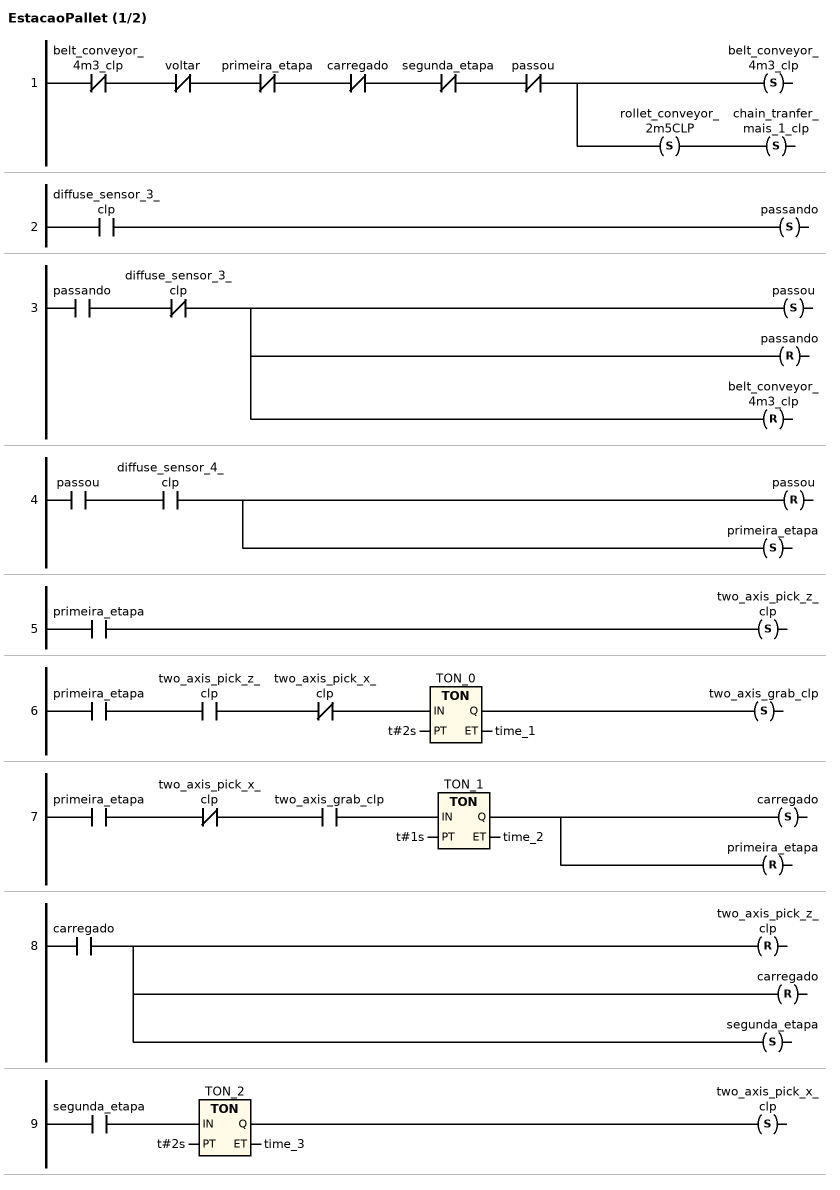
// NETWORK 1
_w1 := NOT belt_conveyor_4m3_clp AND NOT voltar AND NOT primeira_etapa AND NOT carregado AND NOT segunda_etapa AND NOT passou;
belt_conveyor_4m3_clp S= _w1;
rollet_conveyor_2m5CLP S= _w1;
chain_tranfer_mais_1_clp S= _w1;

// NETWORK 2
passando S= diffuse_sensor_3_clp;

// NETWORK 3
_w2 := passando AND NOT diffuse_sensor_3_clp;
passou S= _w2;
passando R= _w2;
belt_conveyor_4m3_clp R= _w2;

// NETWORK 4
_w3 := passou AND diffuse_sensor_4_clp;
passou R= _w3;
primeira_etapa S= _w3;

// NETWORK 5
two_axis_pick_z_clp S= primeira_etapa;

// NETWORK 6
TON_0(IN := primeira_etapa AND two_axis_pick_z_clp AND NOT two_axis_pick_x_clp, PT := t#2s, ET => time_1); // TON
two_axis_grab_clp S= TON_0.Q;

// NETWORK 7
TON_1(IN := primeira_etapa AND NOT two_axis_pick_x_clp AND two_axis_grab_clp, PT := t#1s, ET => time_2); // TON
carregado S= TON_1.Q;
primeira_etapa R= TON_1.Q;

// NETWORK 8
_w4 := carregado;
two_axis_pick_z_clp R= _w4;
carregado R= _w4;
segunda_etapa S= _w4;

// NETWORK 9
TON_2(IN := segunda_etapa, PT := t#2s, ET => time_3); // TON
two_axis_pick_x_clp S= TON_2.Q;

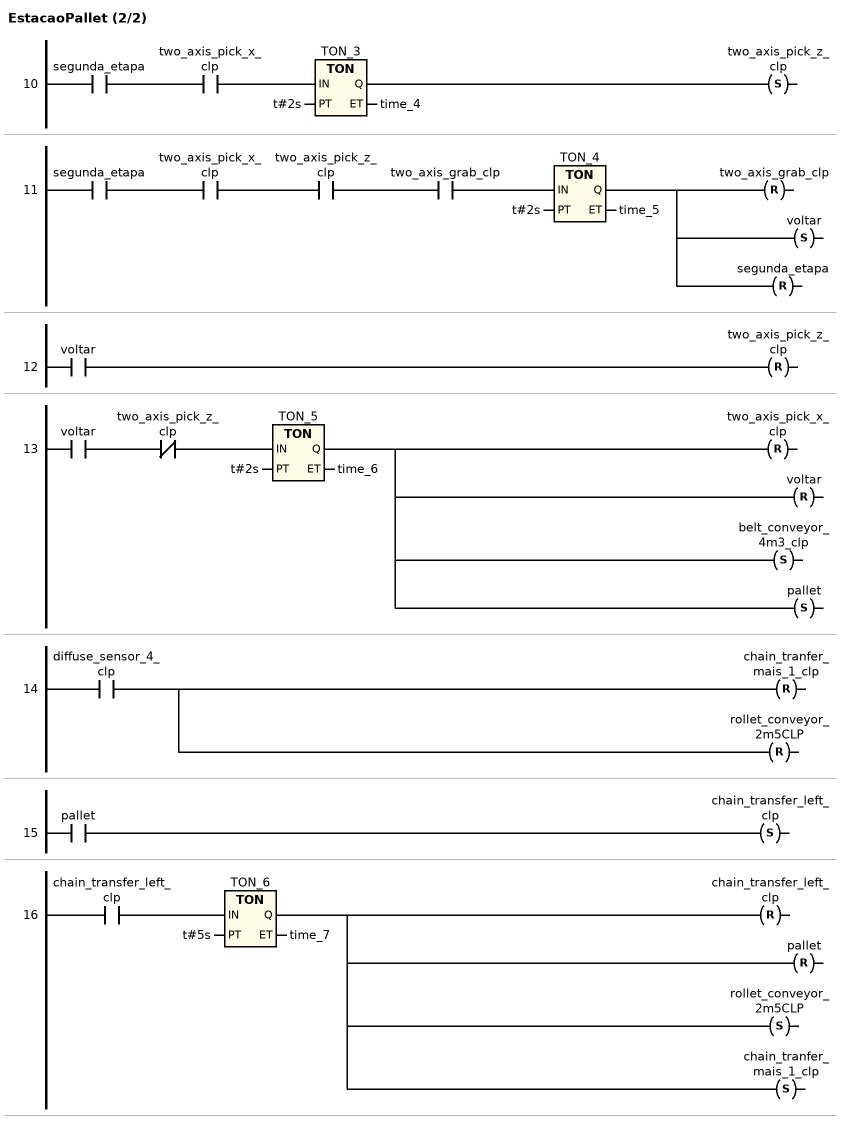
// NETWORK 10
TON_3(IN := segunda_etapa AND two_axis_pick_x_clp, PT := t#2s, ET => time_4); // TON
two_axis_pick_z_clp S= TON_3.Q;

// NETWORK 11
TON_4(
    IN := segunda_etapa AND two_axis_pick_x_clp AND two_axis_pick_z_clp AND two_axis_grab_clp,
    PT := t#2s,
    ET => time_5); // TON
two_axis_grab_clp R= TON_4.Q;
voltar S= TON_4.Q;
segunda_etapa R= TON_4.Q;

// NETWORK 12
two_axis_pick_z_clp R= voltar;

// NETWORK 13
TON_5(IN := voltar AND NOT two_axis_pick_z_clp, PT := t#2s, ET => time_6); // TON
two_axis_pick_x_clp R= TON_5.Q;
voltar R= TON_5.Q;
belt_conveyor_4m3_clp S= TON_5.Q;
pallet S= TON_5.Q;

// NETWORK 14
chain_tranfer_mais_1_clp R= diffuse_sensor_4_clp;
rollet_conveyor_2m5CLP R= diffuse_sensor_4_clp;

// NETWORK 15
chain_transfer_left_clp S= pallet;

// NETWORK 16
TON_6(IN := chain_transfer_left_clp, PT := t#5s, ET => time_7); // TON
chain_transfer_left_clp R= TON_6.Q;
pallet R= TON_6.Q;
rollet_conveyor_2m5CLP S= TON_6.Q;
chain_tranfer_mais_1_clp S= TON_6.Q;

END_PROGRAM

// PLC_PRG_1
PROGRAM PLC_PRG_1
VAR
	passando: BOOL;
	diffuse_sensor_3_clp: BOOL;
	passou: BOOL;
	belt_conveyor_3_clp: BOOL;
	two_axis_pick_z_clp: BOOL;
	two_axis_pick_x_clp: BOOL;
	TON_0: TON;
	time_1: TIME;
	two_axis_grab_clp: BOOL;
	TON_1: TON;
	time_2: TIME;
	carregado: BOOL;
	segunda_etapa: BOOL;
	TON_2: TON;
	time_3: TIME;
	TON_3: TON;
	time_4: TIME;
	TON_4: TON;
	time_5: TIME;
	voltar: BOOL;
	primeira_etapa: BOOL;
	TON_5: TON;
	time_6: TIME;
	pallet: BOOL;
	chain_tranfer_mais_1_clp: BOOL;
	diffuse_sensor_4_clp: BOOL;
	chain_transfer_left_clp: BOOL;
	TON_6: TON;
	time_7: TIME;
END_VAR
VAR // added by the converter: edge detectors and wires of the graphical bodies
    _w1, _w2, _w3, _w4 : BOOL;
END_VAR

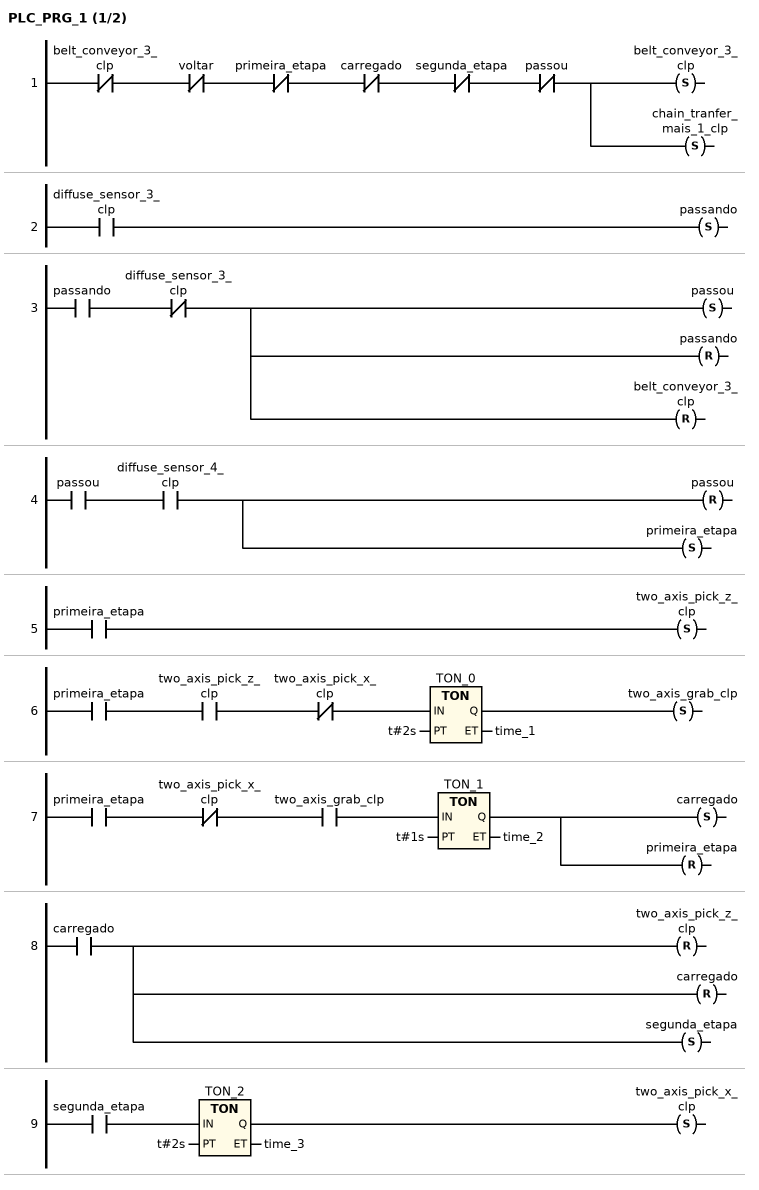
// NETWORK 1
_w1 := NOT belt_conveyor_3_clp AND NOT voltar AND NOT primeira_etapa AND NOT carregado AND NOT segunda_etapa AND NOT passou;
belt_conveyor_3_clp S= _w1;
chain_tranfer_mais_1_clp S= _w1;

// NETWORK 2
passando S= diffuse_sensor_3_clp;

// NETWORK 3
_w2 := passando AND NOT diffuse_sensor_3_clp;
passou S= _w2;
passando R= _w2;
belt_conveyor_3_clp R= _w2;

// NETWORK 4
_w3 := passou AND diffuse_sensor_4_clp;
passou R= _w3;
primeira_etapa S= _w3;

// NETWORK 5
two_axis_pick_z_clp S= primeira_etapa;

// NETWORK 6
TON_0(IN := primeira_etapa AND two_axis_pick_z_clp AND NOT two_axis_pick_x_clp, PT := t#2s, ET => time_1); // TON
two_axis_grab_clp S= TON_0.Q;

// NETWORK 7
TON_1(IN := primeira_etapa AND NOT two_axis_pick_x_clp AND two_axis_grab_clp, PT := t#1s, ET => time_2); // TON
carregado S= TON_1.Q;
primeira_etapa R= TON_1.Q;

// NETWORK 8
_w4 := carregado;
two_axis_pick_z_clp R= _w4;
carregado R= _w4;
segunda_etapa S= _w4;

// NETWORK 9
TON_2(IN := segunda_etapa, PT := t#2s, ET => time_3); // TON
two_axis_pick_x_clp S= TON_2.Q;

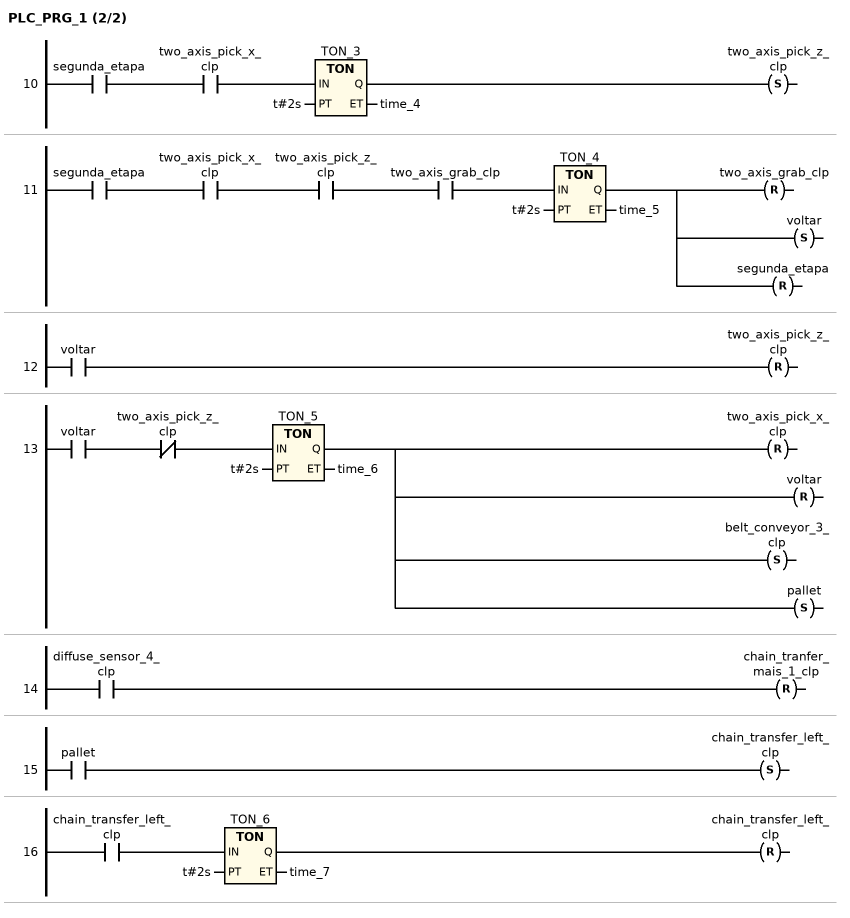
// NETWORK 10
TON_3(IN := segunda_etapa AND two_axis_pick_x_clp, PT := t#2s, ET => time_4); // TON
two_axis_pick_z_clp S= TON_3.Q;

// NETWORK 11
TON_4(
    IN := segunda_etapa AND two_axis_pick_x_clp AND two_axis_pick_z_clp AND two_axis_grab_clp,
    PT := t#2s,
    ET => time_5); // TON
two_axis_grab_clp R= TON_4.Q;
voltar S= TON_4.Q;
segunda_etapa R= TON_4.Q;

// NETWORK 12
two_axis_pick_z_clp R= voltar;

// NETWORK 13
TON_5(IN := voltar AND NOT two_axis_pick_z_clp, PT := t#2s, ET => time_6); // TON
two_axis_pick_x_clp R= TON_5.Q;
voltar R= TON_5.Q;
belt_conveyor_3_clp S= TON_5.Q;
pallet S= TON_5.Q;

// NETWORK 14
chain_tranfer_mais_1_clp R= diffuse_sensor_4_clp;

// NETWORK 15
chain_transfer_left_clp S= pallet;

// NETWORK 16
TON_6(IN := chain_transfer_left_clp, PT := t#2s, ET => time_7); // TON
chain_transfer_left_clp R= TON_6.Q;

END_PROGRAM

// PLC_PRG
PROGRAM PLC_PRG
VAR
	passando: BOOL;
	diffuse_sensor_3_clp: BOOL;
	passou: BOOL;
	belt_conveyor_3_clp: BOOL;
	two_axis_pick_z_clp: BOOL;
	two_axis_pick_x_clp: BOOL;
	TON_0: TON;
	time_1: TIME;
	two_axis_grab_clp: BOOL;
	TON_1: TON;
	time_2: TIME;
	carregado: BOOL;
	segunda_etapa: BOOL;
	TON_2: TON;
	time_3: TIME;
	TON_3: TON;
	time_4: TIME;
	TON_4: TON;
	time_5: TIME;
	voltar: BOOL;
	primeira_etapa: BOOL;
	TON_5: TON;
	time_6: TIME;
	pallet: BOOL;
	chain_tranfer_mais_1_clp: BOOL;
	diffuse_sensor_4_clp: BOOL;
	chain_transfer_left_clp: BOOL;
	TON_6: TON;
	time_7: TIME;
END_VAR
VAR // added by the converter: edge detectors and wires of the graphical bodies
    _w1, _w2, _w3, _w4 : BOOL;
END_VAR

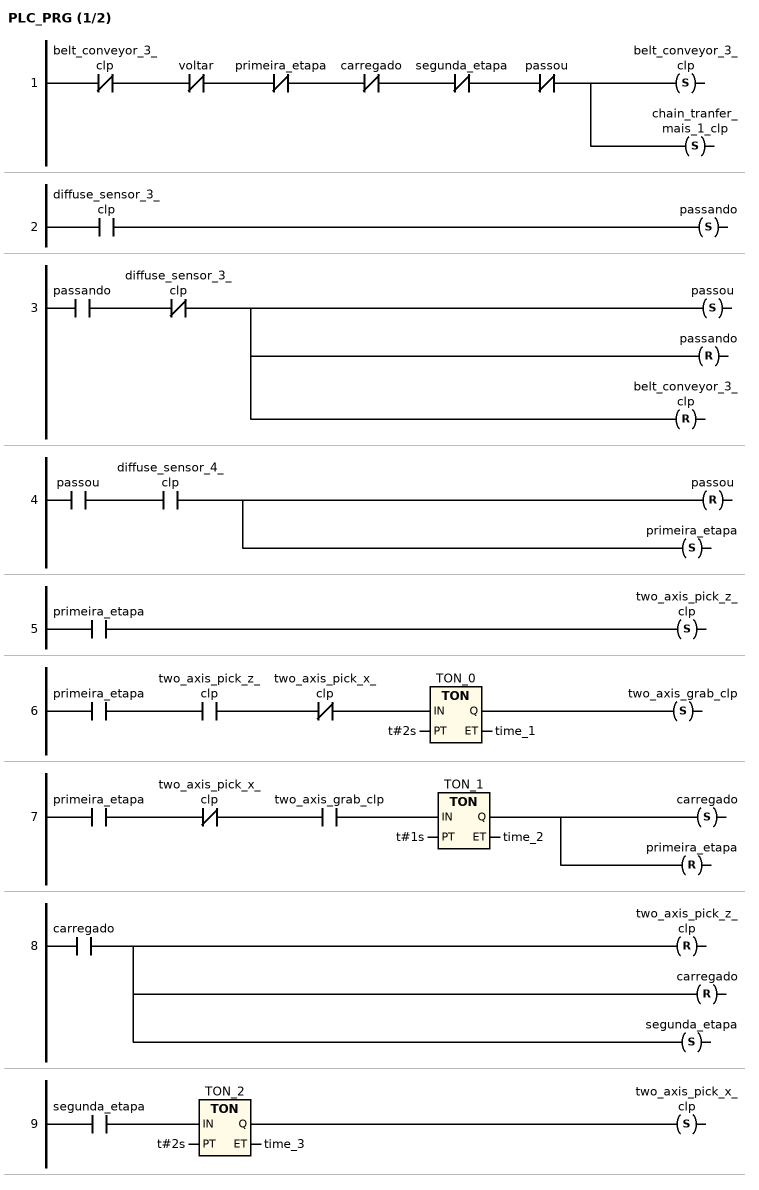
// NETWORK 1
_w1 := NOT belt_conveyor_3_clp AND NOT voltar AND NOT primeira_etapa AND NOT carregado AND NOT segunda_etapa AND NOT passou;
belt_conveyor_3_clp S= _w1;
chain_tranfer_mais_1_clp S= _w1;

// NETWORK 2
passando S= diffuse_sensor_3_clp;

// NETWORK 3
_w2 := passando AND NOT diffuse_sensor_3_clp;
passou S= _w2;
passando R= _w2;
belt_conveyor_3_clp R= _w2;

// NETWORK 4
_w3 := passou AND diffuse_sensor_4_clp;
passou R= _w3;
primeira_etapa S= _w3;

// NETWORK 5
two_axis_pick_z_clp S= primeira_etapa;

// NETWORK 6
TON_0(IN := primeira_etapa AND two_axis_pick_z_clp AND NOT two_axis_pick_x_clp, PT := t#2s, ET => time_1); // TON
two_axis_grab_clp S= TON_0.Q;

// NETWORK 7
TON_1(IN := primeira_etapa AND NOT two_axis_pick_x_clp AND two_axis_grab_clp, PT := t#1s, ET => time_2); // TON
carregado S= TON_1.Q;
primeira_etapa R= TON_1.Q;

// NETWORK 8
_w4 := carregado;
two_axis_pick_z_clp R= _w4;
carregado R= _w4;
segunda_etapa S= _w4;

// NETWORK 9
TON_2(IN := segunda_etapa, PT := t#2s, ET => time_3); // TON
two_axis_pick_x_clp S= TON_2.Q;

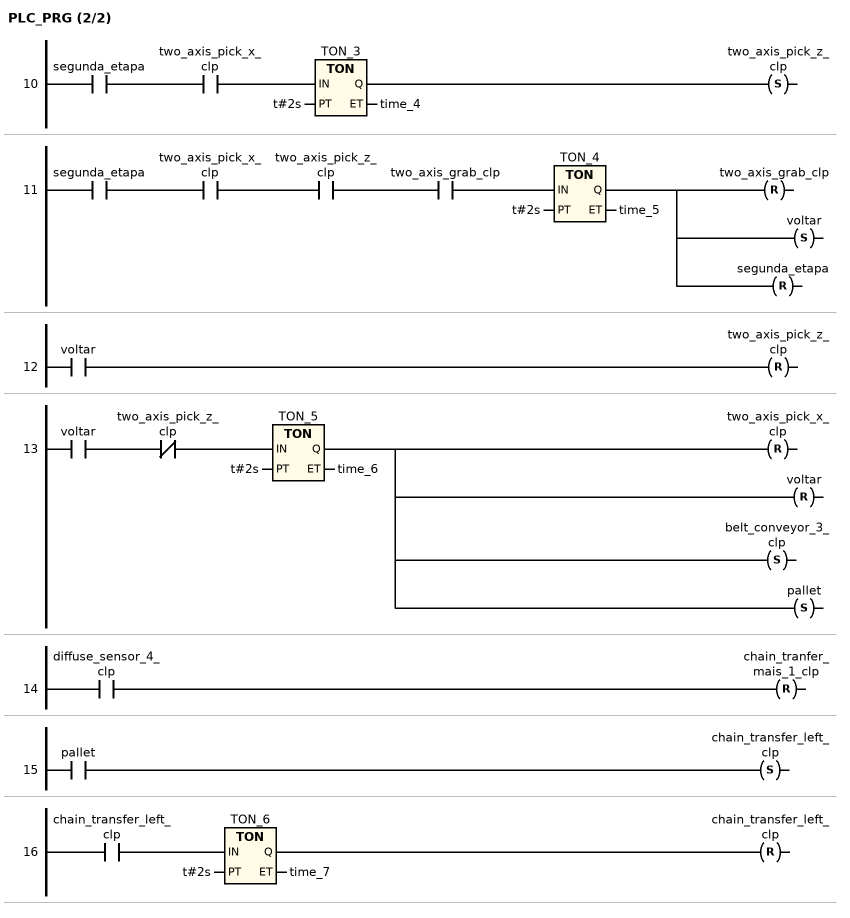
// NETWORK 10
TON_3(IN := segunda_etapa AND two_axis_pick_x_clp, PT := t#2s, ET => time_4); // TON
two_axis_pick_z_clp S= TON_3.Q;

// NETWORK 11
TON_4(
    IN := segunda_etapa AND two_axis_pick_x_clp AND two_axis_pick_z_clp AND two_axis_grab_clp,
    PT := t#2s,
    ET => time_5); // TON
two_axis_grab_clp R= TON_4.Q;
voltar S= TON_4.Q;
segunda_etapa R= TON_4.Q;

// NETWORK 12
two_axis_pick_z_clp R= voltar;

// NETWORK 13
TON_5(IN := voltar AND NOT two_axis_pick_z_clp, PT := t#2s, ET => time_6); // TON
two_axis_pick_x_clp R= TON_5.Q;
voltar R= TON_5.Q;
belt_conveyor_3_clp S= TON_5.Q;
pallet S= TON_5.Q;

// NETWORK 14
chain_tranfer_mais_1_clp R= diffuse_sensor_4_clp;

// NETWORK 15
chain_transfer_left_clp S= pallet;

// NETWORK 16
TON_6(IN := chain_transfer_left_clp, PT := t#2s, ET => time_7); // TON
chain_transfer_left_clp R= TON_6.Q;

END_PROGRAM

// PLC_PRG_2
PROGRAM PLC_PRG_2
VAR
	RollerConveyot2m2CLP: BOOL;
	VisionSensor5CLP: BOOL;
	azul: BOOL;
	TunableBackLimitCLP: BOOL;
	TunableRollmaisCLP: BOOL;
	TunableFrontLimitCLP: BOOL;
	TunableTurnCLP: BOOL;
	TON_0: TON;
	time_1: TIME;
	descarregar: BOOL;
	TON_1: TON;
	time_2: TIME;
END_VAR

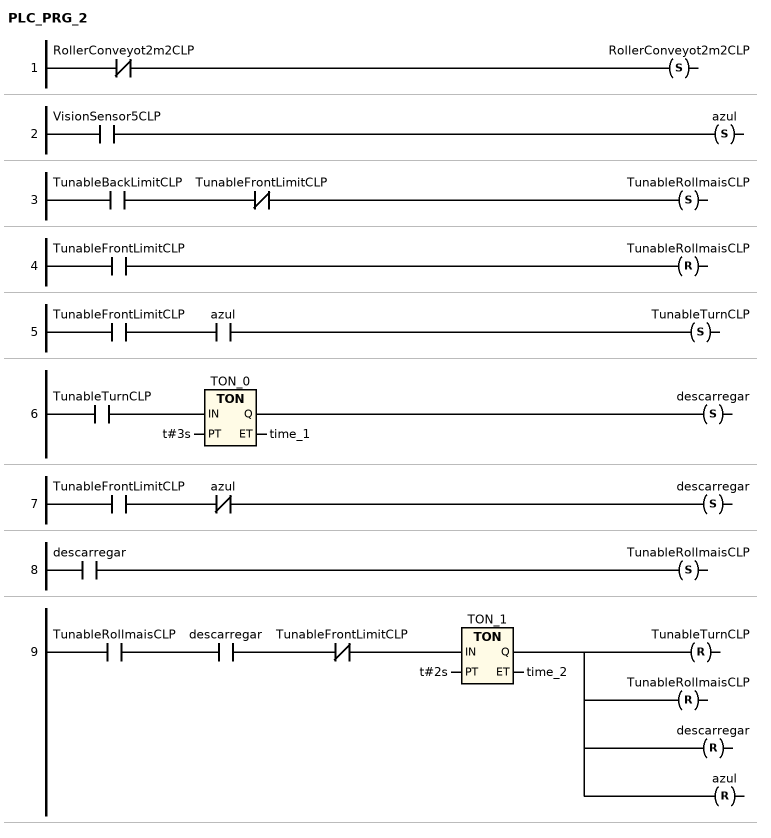
// NETWORK 1
RollerConveyot2m2CLP S= NOT RollerConveyot2m2CLP;

// NETWORK 2
azul S= VisionSensor5CLP;

// NETWORK 3
TunableRollmaisCLP S= TunableBackLimitCLP AND NOT TunableFrontLimitCLP;

// NETWORK 4
TunableRollmaisCLP R= TunableFrontLimitCLP;

// NETWORK 5
TunableTurnCLP S= TunableFrontLimitCLP AND azul;

// NETWORK 6
TON_0(IN := TunableTurnCLP, PT := t#3s, ET => time_1); // TON
descarregar S= TON_0.Q;

// NETWORK 7
descarregar S= TunableFrontLimitCLP AND NOT azul;

// NETWORK 8
TunableRollmaisCLP S= descarregar;

// NETWORK 9
TON_1(IN := TunableRollmaisCLP AND descarregar AND NOT TunableFrontLimitCLP, PT := t#2s, ET => time_2); // TON
TunableTurnCLP R= TON_1.Q;
TunableRollmaisCLP R= TON_1.Q;
descarregar R= TON_1.Q;
azul R= TON_1.Q;

END_PROGRAM

// Device/Application/Teste
PROGRAM Teste
VAR
	RollerConveyot2m2CLP: BOOL;
	VisionSensor5CLP: BOOL;
	azul: BOOL;
	TunableBackLimitCLP: BOOL;
	TunableRollmaisCLP: BOOL;
	TunableFrontLimitCLP: BOOL;
	TunableTurnCLP: BOOL;
	TON_0: TON;
	time_1: TIME;
	descarregar: BOOL;
	TON_1: TON;
	time_2: TIME;
	TesteCLP: BOOL;
	Nada: BOOL;
END_VAR

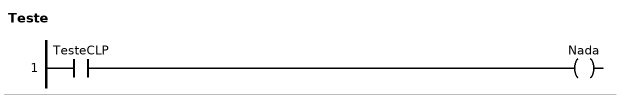
// NETWORK 1
Nada := TesteCLP;

END_PROGRAM
